TYPE ST_PhaseInfo :
STRUCT
  Voltage : REAL;
  Current : REAL;
END_STRUCT
END_TYPE

(* stored: Version 1.1.0.1, ProductVersion 3.1.4024.12
   DUT ST_PhaseInfo: Id {d168336f-9530-4a8f-83f3-12a4e216214e} *)
